SUBAPPLICATION Uebung_012c_sub_AX (* Numeric Value Input und Speichern INI mit Subapp (Adapter Version) *)
  (* Standard: 61499-2; Description: Copyright (c) 2026 Meisterschulen am Ostbahnhof This program and the accompanying materials are made available under the terms of the Eclipse Public License 2.0 which is available at https://www.eclipse.org/legal/epl-2.0/ SPDX-License-Identifier: EPL-2.0 *)
  (* Version 1.0, 2026-04-24, Franz Höpfinger, Meisterschulen am Ostbahnhof, initial API and implementation (AX version) *)
  PACKAGE Uebungen;
  IMPORT isobus::UT::Q::const::IDs::ID_NULL;
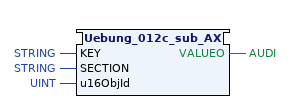
  VAR_INPUT
    KEY : STRING;
    SECTION : STRING;
    u16ObjId : UINT := ID_NULL;
  END_VAR
  PLUGS
    VALUEO : adapter::types::unidirectional::AUDI;
  END_PLUGS
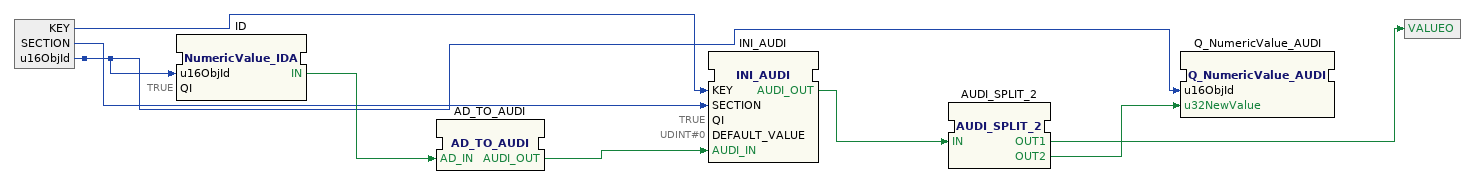
  FBS
    INI_AUDI : eclipse4diac::storage::INI_AUDI(QI := TRUE, DEFAULT_VALUE := UDINT#0);
    ID : isobus::UT::io::NumericValue::NumericValue_IDA(QI := TRUE);
    Q_NumericValue_AUDI : isobus::UT::Q::Q_NumericValue_AUDI;
    AD_TO_AUDI : adapter::conversion::unidirectional::AD_TO_AUDI;
    AUDI_SPLIT_2 : adapter::events::unidirectional::AUDI_SPLIT_2;
  END_FBS
  DATA_CONNECTIONS
    u16ObjId TO Q_NumericValue_AUDI.u16ObjId;
    KEY TO INI_AUDI.KEY;
    SECTION TO INI_AUDI.SECTION;
    u16ObjId TO ID.u16ObjId;
  END_CONNECTIONS
  ADAPTER_CONNECTIONS
    INI_AUDI.AUDI_OUT TO AUDI_SPLIT_2.IN;
    ID.IN TO AD_TO_AUDI.AD_IN;
    AD_TO_AUDI.AUDI_OUT TO INI_AUDI.AUDI_IN;
    AUDI_SPLIT_2.OUT1 TO VALUEO;
    AUDI_SPLIT_2.OUT2 TO Q_NumericValue_AUDI.u32NewValue;
  END_CONNECTIONS
END_SUBAPPLICATION
